TYPE ST_BatchControl :
STRUCT
	bCreate			:BOOL;
	bCancel			:BOOL;
	bOpen			:BOOL;
	bClose			:BOOL;
	bLoad			:BOOL;
	
	sName			:STRING;
	iNumber			:UDINT;
	sProduct		:STRING;
	sComment		:STRING;
	sRecipe			:STRING;
	
	iRecipeType		:INT;
END_STRUCT
END_TYPE

(* stored: Version 1.1.0.1
   DUT ST_BatchControl: Id {d429302e-56cf-4d99-a7b4-0af8f08b8d03} *)
